TYPE SampleTaskFunctionBuffer :
STRUCT
	x : LREAL;
	y : LREAL;
END_STRUCT
END_TYPE

(* stored: Version 1.1.0.1, ProductVersion 3.1.4024.9
   DUT SampleTaskFunctionBuffer: Id {ff0d4e0b-4fe1-0a93-185f-468deeb355e5} *)
